// Mitsubishi GX Works2 project: test_ivrd_ivwr1   PLC: FX3U/FX3UC

PROGRAM MAIN
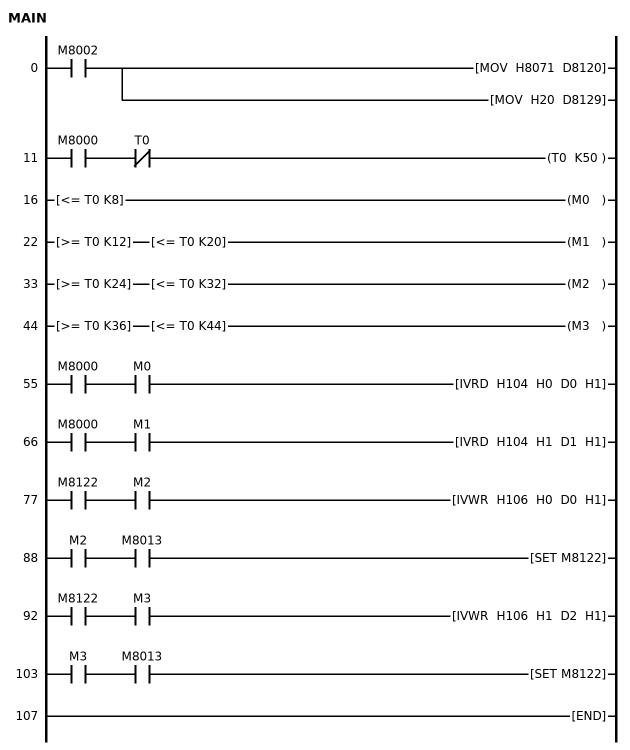
0     LD      M8002
      MOV     H8071 D8120
      MOV     H20 D8129
11    LD      M8000
      ANI     T0
      OUT     T0 K50
16    LD<=    T0 K8
      OUT     M0
22    LD>=    T0 K12
      AND<=   T0 K20
      OUT     M1
33    LD>=    T0 K24
      AND<=   T0 K32
      OUT     M2
44    LD>=    T0 K36
      AND<=   T0 K44
      OUT     M3
55    LD      M8000
      AND     M0
      IVRD    H104 H0 D0 H1
66    LD      M8000
      AND     M1
      IVRD    H104 H1 D1 H1
77    LD      M8122
      AND     M2
      IVWR    H106 H0 D0 H1
88    LD      M2
      AND     M8013
      SET     M8122
92    LD      M8122
      AND     M3
      IVWR    H106 H1 D2 H1
103   LD      M3
      AND     M8013
      SET     M8122
107   END
END_PROGRAM
